// TwinCAT 3 PLC project Untitled1
// ProgramVersion: 3.1.4024.0
// libraries:
//   Tc2_Standard, * (Beckhoff Automation GmbH)
//   Tc2_System, * (Beckhoff Automation GmbH)
//   Tc3_Module, * (Beckhoff Automation GmbH)
// project tree:
//   DUTs/ E_ComponentState.TcTLEO, E_ComponentMode.TcTLEO (not stored)
//   / PlcTask.TcTTO (not stored)
//   POUs/ FB_InductiveSensor.TcPOU, I_Component.TcIO, MAIN.TcPOU (not stored)
// real-time tasks:
//   TASK PlcTask: cycle T#10ms, priority 20, ADS port 350

// ---- DUTs/E_ComponentState.TcTLEO
{attribute 'qualified_only'}
{attribute 'strict'}
TYPE E_ComponentState :
(
	READY 	:= 0,
	BUSY	:= 1,
	DONE	:= 2
);
END_TYPE

// ---- POUs/I_Component.TcIO
INTERFACE I_Component
VAR_INPUT
	sName			: STRING[20];
	bEnable     	: BOOL;
	bStart      	: BOOL;
	bHalt			: BOOL;
	bStop       	: BOOL;
	eMode       	: E_ComponentMode; 		// 0=OFF, 1=AUTO, 2=MANUAL
END_VAR

VAR_OUTPUT
	eState			: E_ComponentState;		// 0=READY, 1=BUSY, 2=DONE
	iErrorCode		: INT;
	sStatusText 	: STRING[50];
END_VAR

METHOD Halt : BOOL
VAR_INPUT
END_VAR
END_METHOD

METHOD Start : BOOL
VAR_INPUT
END_VAR
END_METHOD

METHOD Stop : BOOL
VAR_INPUT
END_VAR
END_METHOD

END_INTERFACE

// ---- POUs/FB_InductiveSensor.TcPOU
// function block for inductive sensor with the option of debouncing + rising and falling edge detection.
FUNCTION_BLOCK FB_InductiveSensor IMPLEMENTS  I_Component
VAR_INPUT
	bSignal			: BOOL;		// Raw input sensor
	tDebounce		: TIME;		// Debounce time
// Interface vars
	sName			: STRING[20];
	bEnable     	: BOOL;
	bStart      	: BOOL;
	bHalt			: BOOL;
	bStop       	: BOOL;
	eMode       	: E_ComponentMode; 		// 0=OFF, 1=AUTO, 2=MANUAL	
END_VAR

VAR_OUTPUT
	bActive			: BOOL;
	bRising			: BOOL;
	bFalling		: BOOL;
// interface vars
	eState			: E_ComponentState;		// 0=READY, 1=BUSY, 2=DONE
	iErrorCode		: INT;
	sStatusText 	: STRING[50];
END_VAR

VAR
	bLastSignal		: BOOL;
	tDebTimer		: TON;
	bSignalStable	: BOOL;
END_VAR

IF bEnable THEN
	IF bLastSignal <> bSignal THEN
		tDebTimer(IN := TRUE, PT := tDebounce);
		eState := E_ComponentState.BUSY;
	ELSE
		tDebTimer(IN := FALSE);
	END_IF
	
	IF tDebTimer.Q THEN
		bSignalStable 	:= bSignal;
		bLastSignal 	:= bSignal;
		eState := E_ComponentState.READY;
	END_IF
	
	bRising		:= (bSignalStable AND NOT bActive);
	bFalling	:= (NOT bSignalStable AND bActive);
	bActive 	:= bSignalStable;
ELSE
	bActive 	:= FALSE;
	bRising		:= FALSE;
	bFalling	:= FALSE;
	tDebTimer(IN := FALSE);
END_IF

METHOD Halt : BOOL
END_METHOD

METHOD Read : BOOL
Read := bSensor;
END_METHOD

METHOD Start : BOOL
END_METHOD

METHOD Stop : BOOL
END_METHOD

END_FUNCTION_BLOCK
